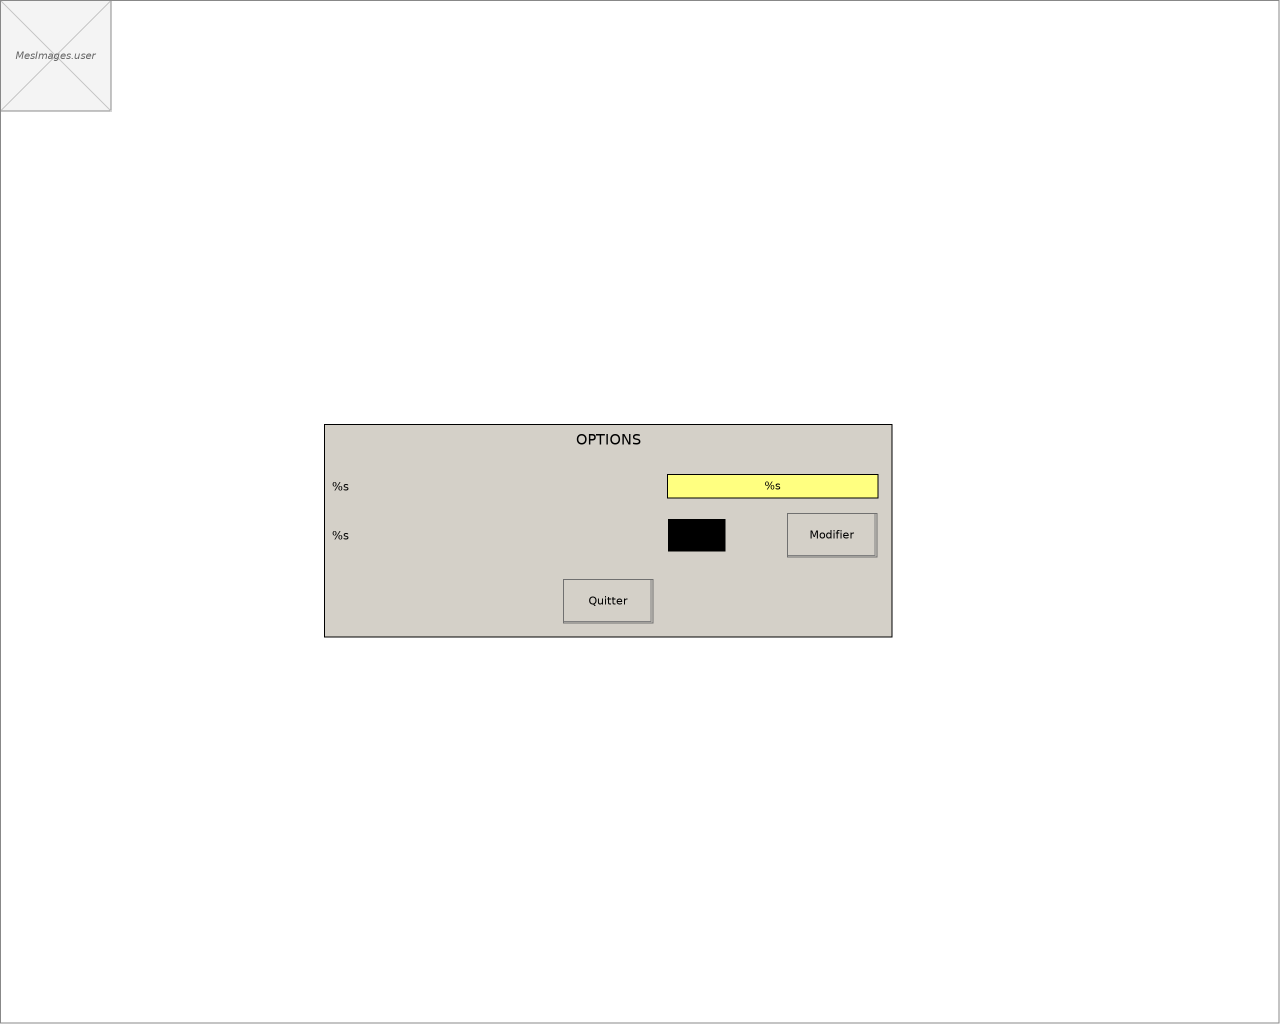
VISUALIZATION UTIL_OPT  // 1280x1024
    Image (0,0 111x111), image: MesImages.user
    RoundedRectangle (324,424 568x213)
    Rectangle (346,425 525x29), "OPTIONS"
    Button (563,579 90x44), "Quitter"
        toggle RQ_PARAM_SYSTEM
        OnMouseClick: change screen: UTIL_MENU
    Rectangle (329,472 295x29), "%s", text list: 'TextList_Users_Menu', text index: 30
    Rectangle (667,474 211x24), "%s", text variable: PRG_USER.TIM_LOGOUT
        OnMouseClick: write the text variable via InputWithLimits
    Rectangle (329,521 295x29), "%s", text list: 'TextList_Users_Menu', text index: 31
    Rectangle (668,519 57x32), "Oui", colour toggle: PRG_USER.OPT_LOGOUT
    Button (787,513 90x44), "Modifier"
        toggle PRG_USER.OPT_LOGOUT
END_VISUALIZATION

(* stored: Version 1.1.0.1, ProductVersion 3.1.4024.10
   Visu UTIL_OPT: Id {4c2b2fd6-384c-4428-95ca-43cdf5240a57} *)
